# EPICS substitutions: pacman-softIoc/pacman_food.subs
file pacman_food.template
{ pattern
  { NAME,	X,	Y , VALX, VALY, FOODSTATE }
  { PACMAN, 1, 1, 31, 31, 1 }
  { PACMAN, 2, 1, 63, 31, 1 }
  { PACMAN, 3, 1, 95, 31, 1 }
  { PACMAN, 4, 1, 127, 31, 1 }
  { PACMAN, 5, 1, 159, 31, 1 }
  { PACMAN, 6, 1, 191, 31, 1 }
  { PACMAN, 7, 1, 223, 31, 1 }
  { PACMAN, 8, 1, 255, 31, 1 }
  { PACMAN, 9, 1, 287, 31, 1 }
  { PACMAN, 10, 1, 319, 31, 1 }
  { PACMAN, 11, 1, 351, 31, 1 }
  { PACMAN, 12, 1, 383, 31, 1 }
  { PACMAN, 13, 1, 479, 31, 1 }
  { PACMAN, 14, 1, 511, 31, 1 }
  { PACMAN, 15, 1, 543, 31, 1 }
  { PACMAN, 16, 1, 575, 31, 1 }
  { PACMAN, 17, 1, 607, 31, 1 }
  { PACMAN, 18, 1, 639, 31, 1 }
  { PACMAN, 19, 1, 671, 31, 1 }
  { PACMAN, 20, 1, 703, 31, 1 }
  { PACMAN, 21, 1, 735, 31, 1 }
  { PACMAN, 22, 1, 767, 31, 1 }
  { PACMAN, 23, 1, 799, 31, 1 }
  { PACMAN, 24, 1, 831, 31, 1 }
  { PACMAN, 25, 1, 31, 63, 1 }
  { PACMAN, 26, 1, 191, 63, 1 }
  { PACMAN, 27, 1, 383, 63, 1 }
  { PACMAN, 28, 1, 479, 63, 1 }
  { PACMAN, 1, 2, 671, 63, 1 }
  { PACMAN, 2, 2, 831, 63, 1 }
  { PACMAN, 3, 2, 31, 95, 2 }
  { PACMAN, 4, 2, 191, 95, 1 }
  { PACMAN, 5, 2, 383, 95, 1 }
  { PACMAN, 6, 2, 479, 95, 1 }
  { PACMAN, 7, 2, 671, 95, 1 }
  { PACMAN, 8, 2, 831, 95, 2 }
  { PACMAN, 9, 2, 31, 127, 1 }
  { PACMAN, 10, 2, 191, 127, 1 }
  { PACMAN, 11, 2, 383, 127, 1 }
  { PACMAN, 12, 2, 479, 127, 1 }
  { PACMAN, 13, 2, 671, 127, 1 }
  { PACMAN, 14, 2, 831, 127, 1 }
  { PACMAN, 15, 2, 31, 159, 1 }
  { PACMAN, 16, 2, 63, 159, 1 }
  { PACMAN, 17, 2, 95, 159, 1 }
  { PACMAN, 18, 2, 127, 159, 1 }
  { PACMAN, 19, 2, 159, 159, 1 }
  { PACMAN, 20, 2, 191, 159, 1 }
  { PACMAN, 21, 2, 223, 159, 1 }
  { PACMAN, 22, 2, 255, 159, 1 }
  { PACMAN, 23, 2, 287, 159, 1 }
  { PACMAN, 24, 2, 319, 159, 1 }
  { PACMAN, 25, 2, 351, 159, 1 }
  { PACMAN, 26, 2, 383, 159, 1 }
  { PACMAN, 27, 2, 415, 159, 1 }
  { PACMAN, 28, 2, 447, 159, 1 }
  { PACMAN, 1, 3, 479, 159, 1 }
  { PACMAN, 2, 3, 511, 159, 1 }
  { PACMAN, 3, 3, 543, 159, 1 }
  { PACMAN, 4, 3, 575, 159, 1 }
  { PACMAN, 5, 3, 607, 159, 1 }
  { PACMAN, 6, 3, 639, 159, 1 }
  { PACMAN, 7, 3, 671, 159, 1 }
  { PACMAN, 8, 3, 703, 159, 1 }
  { PACMAN, 9, 3, 735, 159, 1 }
  { PACMAN, 10, 3, 767, 159, 1 }
  { PACMAN, 11, 3, 799, 159, 1 }
  { PACMAN, 12, 3, 831, 159, 1 }
  { PACMAN, 13, 3, 31, 191, 1 }
  { PACMAN, 14, 3, 191, 191, 1 }
  { PACMAN, 15, 3, 287, 191, 1 }
  { PACMAN, 16, 3, 575, 191, 1 }
  { PACMAN, 17, 3, 671, 191, 1 }
  { PACMAN, 18, 3, 831, 191, 1 }
  { PACMAN, 19, 3, 31, 223, 1 }
  { PACMAN, 20, 3, 191, 223, 1 }
  { PACMAN, 21, 3, 287, 223, 1 }
  { PACMAN, 22, 3, 575, 223, 1 }
  { PACMAN, 23, 3, 671, 223, 1 }
  { PACMAN, 24, 3, 831, 223, 1 }
  { PACMAN, 25, 3, 31, 255, 1 }
  { PACMAN, 26, 3, 63, 255, 1 }
  { PACMAN, 27, 3, 95, 255, 1 }
  { PACMAN, 28, 3, 127, 255, 1 }
  { PACMAN, 1, 4, 159, 255, 1 }
  { PACMAN, 2, 4, 191, 255, 1 }
  { PACMAN, 3, 4, 287, 255, 1 }
  { PACMAN, 4, 4, 319, 255, 1 }
  { PACMAN, 5, 4, 351, 255, 1 }
  { PACMAN, 6, 4, 383, 255, 1 }
  { PACMAN, 7, 4, 479, 255, 1 }
  { PACMAN, 8, 4, 511, 255, 1 }
  { PACMAN, 9, 4, 543, 255, 1 }
  { PACMAN, 10, 4, 575, 255, 1 }
  { PACMAN, 11, 4, 671, 255, 1 }
  { PACMAN, 12, 4, 703, 255, 1 }
  { PACMAN, 13, 4, 735, 255, 1 }
  { PACMAN, 14, 4, 767, 255, 1 }
  { PACMAN, 15, 4, 799, 255, 1 }
  { PACMAN, 16, 4, 831, 255, 1 }
  { PACMAN, 17, 4, 191, 287, 1 }
  { PACMAN, 18, 4, 671, 287, 1 }
  { PACMAN, 19, 4, 191, 319, 1 }
  { PACMAN, 20, 4, 671, 319, 1 }
  { PACMAN, 21, 4, 191, 351, 1 }
  { PACMAN, 22, 4, 671, 351, 1 }
  { PACMAN, 23, 4, 191, 383, 1 }
  { PACMAN, 24, 4, 671, 383, 1 }
  { PACMAN, 25, 4, 191, 415, 1 }
  { PACMAN, 26, 4, 671, 415, 1 }
  { PACMAN, 27, 4, 191, 447, 1 }
  { PACMAN, 28, 4, 671, 447, 1 }
  { PACMAN, 1, 5, 191, 479, 1 }
  { PACMAN, 2, 5, 671, 479, 1 }
  { PACMAN, 3, 5, 191, 511, 1 }
  { PACMAN, 4, 5, 671, 511, 1 }
  { PACMAN, 5, 5, 191, 543, 1 }
  { PACMAN, 6, 5, 671, 543, 1 }
  { PACMAN, 7, 5, 191, 575, 1 }
  { PACMAN, 8, 5, 671, 575, 1 }
  { PACMAN, 9, 5, 191, 607, 1 }
  { PACMAN, 10, 5, 671, 607, 1 }
  { PACMAN, 11, 5, 31, 639, 1 }
  { PACMAN, 12, 5, 63, 639, 1 }
  { PACMAN, 13, 5, 95, 639, 1 }
  { PACMAN, 14, 5, 127, 639, 1 }
  { PACMAN, 15, 5, 159, 639, 1 }
  { PACMAN, 16, 5, 191, 639, 1 }
  { PACMAN, 17, 5, 223, 639, 1 }
  { PACMAN, 18, 5, 255, 639, 1 }
  { PACMAN, 19, 5, 287, 639, 1 }
  { PACMAN, 20, 5, 319, 639, 1 }
  { PACMAN, 21, 5, 351, 639, 1 }
  { PACMAN, 22, 5, 383, 639, 1 }
  { PACMAN, 23, 5, 479, 639, 1 }
  { PACMAN, 24, 5, 511, 639, 1 }
  { PACMAN, 25, 5, 543, 639, 1 }
  { PACMAN, 26, 5, 575, 639, 1 }
  { PACMAN, 27, 5, 607, 639, 1 }
  { PACMAN, 28, 5, 639, 639, 1 }
  { PACMAN, 1, 6, 671, 639, 1 }
  { PACMAN, 2, 6, 703, 639, 1 }
  { PACMAN, 3, 6, 735, 639, 1 }
  { PACMAN, 4, 6, 767, 639, 1 }
  { PACMAN, 5, 6, 799, 639, 1 }
  { PACMAN, 6, 6, 831, 639, 1 }
  { PACMAN, 7, 6, 31, 671, 1 }
  { PACMAN, 8, 6, 191, 671, 1 }
  { PACMAN, 9, 6, 383, 671, 1 }
  { PACMAN, 10, 6, 479, 671, 1 }
  { PACMAN, 11, 6, 671, 671, 1 }
  { PACMAN, 12, 6, 831, 671, 1 }
  { PACMAN, 13, 6, 31, 703, 1 }
  { PACMAN, 14, 6, 191, 703, 1 }
  { PACMAN, 15, 6, 383, 703, 1 }
  { PACMAN, 16, 6, 479, 703, 1 }
  { PACMAN, 17, 6, 671, 703, 1 }
  { PACMAN, 18, 6, 831, 703, 1 }
  { PACMAN, 19, 6, 31, 735, 2 }
  { PACMAN, 20, 6, 63, 735, 1 }
  { PACMAN, 21, 6, 95, 735, 1 }
  { PACMAN, 22, 6, 191, 735, 1 }
  { PACMAN, 23, 6, 223, 735, 1 }
  { PACMAN, 24, 6, 255, 735, 1 }
  { PACMAN, 25, 6, 287, 735, 1 }
  { PACMAN, 26, 6, 319, 735, 1 }
  { PACMAN, 27, 6, 351, 735, 1 }
  { PACMAN, 28, 6, 383, 735, 1 }
  { PACMAN, 1, 7, 479, 735, 1 }
  { PACMAN, 2, 7, 511, 735, 1 }
  { PACMAN, 3, 7, 543, 735, 1 }
  { PACMAN, 4, 7, 575, 735, 1 }
  { PACMAN, 5, 7, 607, 735, 1 }
  { PACMAN, 6, 7, 639, 735, 1 }
  { PACMAN, 7, 7, 671, 735, 1 }
  { PACMAN, 8, 7, 767, 735, 1 }
  { PACMAN, 9, 7, 799, 735, 1 }
  { PACMAN, 10, 7, 831, 735, 2 }
  { PACMAN, 11, 7, 95, 767, 1 }
  { PACMAN, 12, 7, 191, 767, 1 }
  { PACMAN, 13, 7, 287, 767, 1 }
  { PACMAN, 14, 7, 575, 767, 1 }
  { PACMAN, 15, 7, 671, 767, 1 }
  { PACMAN, 16, 7, 767, 767, 1 }
  { PACMAN, 17, 7, 95, 799, 1 }
  { PACMAN, 18, 7, 191, 799, 1 }
  { PACMAN, 19, 7, 287, 799, 1 }
  { PACMAN, 20, 7, 575, 799, 1 }
  { PACMAN, 21, 7, 671, 799, 1 }
  { PACMAN, 22, 7, 767, 799, 1 }
  { PACMAN, 23, 7, 31, 831, 1 }
  { PACMAN, 24, 7, 63, 831, 1 }
  { PACMAN, 25, 7, 95, 831, 1 }
  { PACMAN, 26, 7, 127, 831, 1 }
  { PACMAN, 27, 7, 159, 831, 1 }
  { PACMAN, 28, 7, 191, 831, 1 }
  { PACMAN, 1, 8, 287, 831, 1 }
  { PACMAN, 2, 8, 319, 831, 1 }
  { PACMAN, 3, 8, 351, 831, 1 }
  { PACMAN, 4, 8, 383, 831, 1 }
  { PACMAN, 5, 8, 479, 831, 1 }
  { PACMAN, 6, 8, 511, 831, 1 }
  { PACMAN, 7, 8, 543, 831, 1 }
  { PACMAN, 8, 8, 575, 831, 1 }
  { PACMAN, 9, 8, 671, 831, 1 }
  { PACMAN, 10, 8, 703, 831, 1 }
  { PACMAN, 11, 8, 735, 831, 1 }
  { PACMAN, 12, 8, 767, 831, 1 }
  { PACMAN, 13, 8, 799, 831, 1 }
  { PACMAN, 14, 8, 831, 831, 1 }
  { PACMAN, 15, 8, 31, 863, 1 }
  { PACMAN, 16, 8, 383, 863, 1 }
  { PACMAN, 17, 8, 479, 863, 1 }
  { PACMAN, 18, 8, 831, 863, 1 }
  { PACMAN, 19, 8, 31, 895, 1 }
  { PACMAN, 20, 8, 383, 895, 1 }
  { PACMAN, 21, 8, 479, 895, 1 }
  { PACMAN, 22, 8, 831, 895, 1 }
  { PACMAN, 23, 8, 31, 927, 1 }
  { PACMAN, 24, 8, 63, 927, 1 }
  { PACMAN, 25, 8, 95, 927, 1 }
  { PACMAN, 26, 8, 127, 927, 1 }
  { PACMAN, 27, 8, 159, 927, 1 }
  { PACMAN, 28, 8, 191, 927, 1 }
  { PACMAN, 1, 9, 223, 927, 1 }
  { PACMAN, 2, 9, 255, 927, 1 }
  { PACMAN, 3, 9, 287, 927, 1 }
  { PACMAN, 4, 9, 319, 927, 1 }
  { PACMAN, 5, 9, 351, 927, 1 }
  { PACMAN, 6, 9, 383, 927, 1 }
  { PACMAN, 7, 9, 415, 927, 1 }
  { PACMAN, 8, 9, 447, 927, 1 }
  { PACMAN, 9, 9, 479, 927, 1 }
  { PACMAN, 10, 9, 511, 927, 1 }
  { PACMAN, 11, 9, 543, 927, 1 }
  { PACMAN, 12, 9, 575, 927, 1 }
  { PACMAN, 13, 9, 607, 927, 1 }
  { PACMAN, 14, 9, 639, 927, 1 }
  { PACMAN, 15, 9, 671, 927, 1 }
  { PACMAN, 16, 9, 703, 927, 1 }
  { PACMAN, 17, 9, 735, 927, 1 }
  { PACMAN, 18, 9, 767, 927, 1 }
  { PACMAN, 19, 9, 799, 927, 1 }
  { PACMAN, 20, 9, 831, 927, 1 }
}
